FUNCTION_BLOCK FB_PowerControlledHeaterContactor EXTENDS FB_Actuator2Point

VAR
	
	//I/O Links	
	bSetStatusOn_OUT 	AT %Q*	: 	BOOL := FALSE;		
	
END_VAR

SelectControlMode();

METHOD SetState_BO : BOOL
VAR_INPUT
END_VAR
//output
bSetStatusOn_OUT := bSetStatusOn;
END_METHOD

END_FUNCTION_BLOCK

(* stored: Version 1.1.0.1, ProductVersion 3.1.4024.6
   POU FB_PowerControlledHeaterContactor: Id {537e7a10-0a68-45e8-b712-1127278d87e0}, SpecialFunc None
   Method SetState_BO: Id {9694878c-e321-4b69-b3b9-7424d792fe2e} *)
